FUNCTION_BLOCK M_GET (* Retrieve a Matrix Element *)
  (* Standard: 61499-1; Classification: Matrix Operations; Function: Initialization *)
  (* Version 0.0, 2002-03-07, JHC, Rockwell Automation *)
  (* Compiler header: package fb.rt.math; *)
  (* Compiler Java IBM VisualAge 3.0 *)
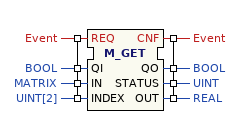
  EVENT_INPUT
    REQ WITH QI, IN, INDEX; (* Retrieve the data at location INDEX *)
  END_EVENT
  EVENT_OUTPUT
    CNF WITH QO, STATUS, OUT;
  END_EVENT
  VAR_INPUT
    QI : BOOL; (* 0=Inhibit,1=Enable *)
    IN : MATRIX; (* Matrix from which to get data *)
    INDEX : ARRAY [0..1] OF UINT; (* [row,column] *)
  END_VAR
  VAR_OUTPUT
    QO : BOOL; (* 1=OK,0=Inhibited or Error *)
    STATUS : UINT; (* 0=OK,1=INHIBITED,13=ARRAY_SIZE_ERROR *)
    OUT : REAL; (* Data at INDEX location of IN *)
  END_VAR
END_FUNCTION_BLOCK
